Yaskawa INFORM job: 66.JBI

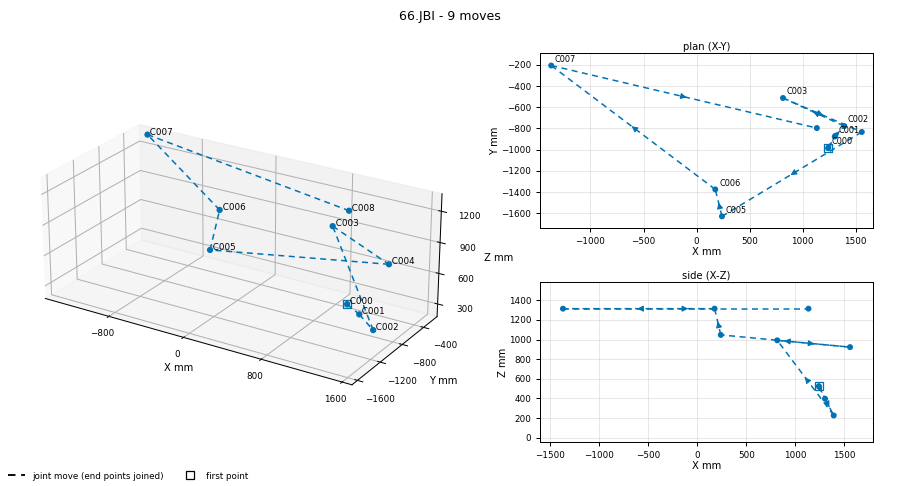
[picture p0: tool path of 66.JBI, 9 of 9 moves have a stored position in this frame; points joined in program order, loops and branches not executed]
/JOB
//NAME 66
//POS
///NPOS 9,0,0,0
///TOOL 0
///RECTAN
///RCONF 1,0,0,0,0
C000=1239.882,-985.527,525.255,95.36,10.58,-67.72
///RCONF 0,0,0,0,0
C001=1302.717,-875.432,397.225,-51.36,48.61,-83.32
C002=1391.582,-777.153,226.180,-42.29,64.66,-71.00
C003=815.094,-512.699,992.809,-150.87,-49.78,-52.58
C004=1557.658,-833.085,923.393,-150.87,-49.78,-52.58
C005=239.464,-1628.244,1047.942,-122.19,-57.25,-120.33
C006=176.499,-1374.262,1315.584,-106.07,-63.67,-134.40
C007=-1370.104,-206.520,1315.549,-106.07,-63.66,136.85
C008=1134.162,-795.935,1315.549,-106.07,-63.66,-86.78
//INST
///DATE 2014/11/09 01:48
///ATTR 0,0,0,0,0,0,0,0,0,0,0,0,1,0,0,0
///FRAME BASE
NOP
*1
PAUSE
MOVJ C000 VJ=100.00 CONT
MOVJ C001 VJ=100.00 CONT
MOVJ C002 VJ=100.00 CONT
MOVJ C003 VJ=100.00 CONT
MOVJ C004 VJ=100.00 CONT
MOVJ C005 VJ=100.00 CONT
MOVJ C006 VJ=100.00 CONT
MOVJ C007 VJ=100.00 CONT
MOVJ C008 VJ=100.00 CONT
JUMP *1
END
